TYPE ST_ProbesSet :
STRUCT
	
	abProbeError							AT %I*			: ARRAY[1..4] OF BOOL;
	anRawMeasurement						AT %I*			: ARRAY[1..4] OF DINT;
	anScaledRawMeasurement									: ARRAY[1..4] OF REAL;
	
END_STRUCT
END_TYPE

(* stored: Version 1.1.0.1, ProductVersion 3.1.4026.17
   DUT ST_ProbesSet: Id {b3bdf078-3dea-4bf0-b516-cc50c4bd1eba} *)
